TYPE ST_RecipeTypeAteqDevice :
STRUCT
	nIdx	: UINT;
	bEnable	: BOOL;
	bEnableAutoZero	: BOOL; // if TRUE Auto Zero runs before each program Start
	nActiveProgramCount	: UINT;
END_STRUCT
END_TYPE

(* stored: Version 1.1.0.1
   DUT ST_RecipeTypeAteqDevice: Id {fc992741-4327-0ae7-0253-1d10a3ce01e7} *)
